FUNCTION_BLOCK PUBLIC GearMoverSequence
VAR_INPUT
	ThisMover : IMover;
	XtsTrack : IXtsTrack;
	StateMachine : IPmlStateMachine;
END_VAR
VAR_OUTPUT
END_VAR
VAR
	axesGear	: GearInCA;
	MoverToGearTo: UDINT;
		State :(
        Init,                                               
        Available,
		MovingToStart, 
		AtStart,                                 
        MovingToStation,
		QueuedAtStation,
		AtStation);  
END_VAR
VAR_IN_OUT
	MoverArray : ARRAY[*] OF IMover;
END_VAR



MoverToGearTo := ThisMover.AxisRef.NcToPlc.AxisId - 1;

axesGear(_MasterAxis := MoverArray[].AxisRef, _SlaveAxis := ThisMover.AxisRef);

METHOD PUBLIC Gear : BOOL
VAR_INPUT
	MasterPosition : MC_LREAL;
	SlavePosition : MC_LREAL;
END_VAR
IF NOT axesGear.Busy THEN
		axesGear.Sync(MasterPosition := MasterPosition, SlavePosition := SlavePosition);
		Gear := TRUE;
END_IF
END_METHOD

END_FUNCTION_BLOCK

(* stored: Version 1.1.0.1, ProductVersion 3.1.4024.9
   POU GearMoverSequence: Id {e1681ea0-a376-4b8a-bd4c-9ec4a0739fe2}, SpecialFunc None
   Method Gear: Id {e70c4ab6-700a-4f7f-96e2-f6bea672eae8} *)
